// TIA Portal V20 export
DATA_BLOCK "SBK02"   // DB208
// stored: MemoryReserve 100
   VAR
      "X1-0 SCS box: SCS mode select, Setup" : Bool;
      "X2-1 SCS box: SCS mode select, Disable" : Bool;
      "X3-2 Frame Corver Detect Sensor" : Bool;
      "X4-3  SAFETY DOOR LOCK7.INPUT" : Bool;
      "X1-4 SCS box: SCS mode select, Auto" : Bool;
      "X2-5 SPARE" : Bool;
      "X3-6 SPARE" : Bool;
      "X4-7 SAFETY DOOR LOCK7.INPUT" : Bool;
      "X5-0 SCS box: Pendant required on, yellow" : Bool;
      "X6-1 SCS box: SCS Disable mode selected, green" : Bool;
      "X7-2 SAFETY DOOR LOCK7.OUTPUT" : Bool;
   END_VAR
BEGIN
END_DATA_BLOCK
